// TIA Portal project "FactoryIO_Template_S7-1200_V16_V16" (V16)
// Vorlageprojekt für das Buch mit Zielsystem S7-1200

(* hardware
DEVICE "S7-1200-Station_1"  S7-1200 Station
   slot 0: "Baugruppenträger_0"  Rack  V1.0
   slot 1: "PLC_1"  CPU 1211C DC/DC/DC  6ES7 211-1AE40-0XB0  V4.1
*)

// ===== PLC "PLC_1"  CPU 1211C DC/DC/DC =====

VAR_GLOBAL   // PLC tag table "Standard-Variablentabelle"
   "START" AT %I0.0 : Bool;
   "STOP" AT %I0.1 : Bool;
   "V.S1" AT %I0.2 : Bool;
   "V.S4" AT %I0.3 : Bool;
   "V.S2" AT %I0.4 : Bool;
   "V.S3" AT %I0.5 : Bool;
   "BELT(6M)1" AT %Q0.0 : Bool;
   "BELT(2M)1" AT %Q0.1 : Bool;
   "BELLT(2M)2" AT %Q0.2 : Bool;
   "BELT(2M)3" AT %Q0.3 : Bool;
   "BELT(2M)4" AT %Q0.4 : Bool;
   "BELT CCW" AT %Q0.5 : Bool;
   "P1" AT %Q0.6 : Bool;
   "MOVE1" AT %Q0.7 : Bool;
   "P2" AT %Q1.0 : Bool;
   "MOVE2" AT %Q1.1 : Bool;
   "P3" AT %Q1.2 : Bool;
   "MOVE3" AT %Q1.3 : Bool;
   "MARKER" AT %M0.0 : Bool;
   "MARKER2" AT %M0.1 : Bool;
   "MARKER3" AT %M0.2 : Bool;
   "MARKER4" AT %M0.3 : Bool;
   "P1 MARKER" AT %M0.4 : Bool;
   "P3 MARKER" AT %M0.5 : Bool;
   "P2 MARKER" AT %M0.6 : Bool;
END_VAR

// folder: System blocks/Program resources

DATA_BLOCK "T1"   // DB1
{ S7_Optimized_Access := 'TRUE' }
AUTHOR : Simatic
FAMILY : IEC
NAME : IEC_TMR
VERSION : 1.0
// stored: InstanceOfName IEC_TIMER
"IEC_TIMER"
BEGIN
END_DATA_BLOCK

DATA_BLOCK "T2"   // DB2
{ S7_Optimized_Access := 'TRUE' }
AUTHOR : Simatic
FAMILY : IEC
NAME : IEC_TMR
VERSION : 1.0
// stored: InstanceOfName IEC_TIMER
"IEC_TIMER"
BEGIN
END_DATA_BLOCK

DATA_BLOCK "T3"   // DB3
{ S7_Optimized_Access := 'TRUE' }
AUTHOR : Simatic
FAMILY : IEC
NAME : IEC_TMR
VERSION : 1.0
// stored: InstanceOfName IEC_TIMER
"IEC_TIMER"
BEGIN
END_DATA_BLOCK

// folder: (top level)

FUNCTION "MHJ-PLC-Lab-Function-S71200" : Void   // FC9000, SCL
{ S7_Optimized_Access := 'TRUE' }
VERSION : 0.1
   VAR_TEMP
      rdTimeReturn : Int;
      outputTime : DTL;
      SyncVal : Byte;
      forVal : Int;
      forVal_2 : Int;
      Value : Byte;
   END_VAR
   VAR CONSTANT
      CompVal : Byte := 16#34;
      Value_01 : Byte := 16#11;
      Value_01_DW : DWord := 16#A165_D992;
      Value_02_DW : DWord := 16#58BE_4401;
   END_VAR
BEGIN

   #Value:=PEEK(area := 16#82,
        dbNumber := 0,
        byteOffset := 511);
   #Value := #Value + 1;

   POKE(area := 16#82,
        dbNumber := 0,
        byteOffset := 511,
        value := #Value);

   POKE(area:=16#81,
        dbNumber:=0,
        byteOffset:=1016,
        value:=#Value_01_DW);
   POKE(area := 16#81,
        dbNumber := 0,
        byteOffset := 1020,
        value := #Value_02_DW);

   POKE(area := 16#81,
        dbNumber := 0,
        byteOffset := 511,
        value := B#16#00);

   FOR #forVal := 0 TO 120 DO
       FOR #forVal_2:=0 TO 10 DO
           #rdTimeReturn:=RD_SYS_T(#outputTime);
           #rdTimeReturn := WR_SYS_T(#outputTime);
           #rdTimeReturn := RD_SYS_T(#outputTime);
           #rdTimeReturn := WR_SYS_T(#outputTime);
       END_FOR;
       #SyncVal:= PEEK(area := 16#81,
                      dbNumber := 0,
                      byteOffset := 511);
       IF #SyncVal = #CompVal THEN
          GOTO M_1;
       END_IF;
   END_FOR;
   RETURN;

   M_1:
   POKE(area := 16#81,
        dbNumber := 0,
        byteOffset := 511,
        value := B#16#0);
END_FUNCTION

ORGANIZATION_BLOCK "Main"   // OB1, LAD, ProgramCycle
TITLE = "Main Program Sweep (Cycle)"
{ S7_Optimized_Access := 'TRUE' }
VERSION : 0.1
   VAR_INPUT
      Initial_Call : Bool;   // Initial call of this OB
      Remanence : Bool;   // =True, if remanent data are available
   END_VAR
BEGIN

REGION Network 1: Konnektierungsbaustein für PLC-Lab
   // Im Netzwerk 1 wird der Konnektierungsbaustein für PLC-Lab aufgerufen.
   // Dieser Aufruf darf nicht entfernt werden!
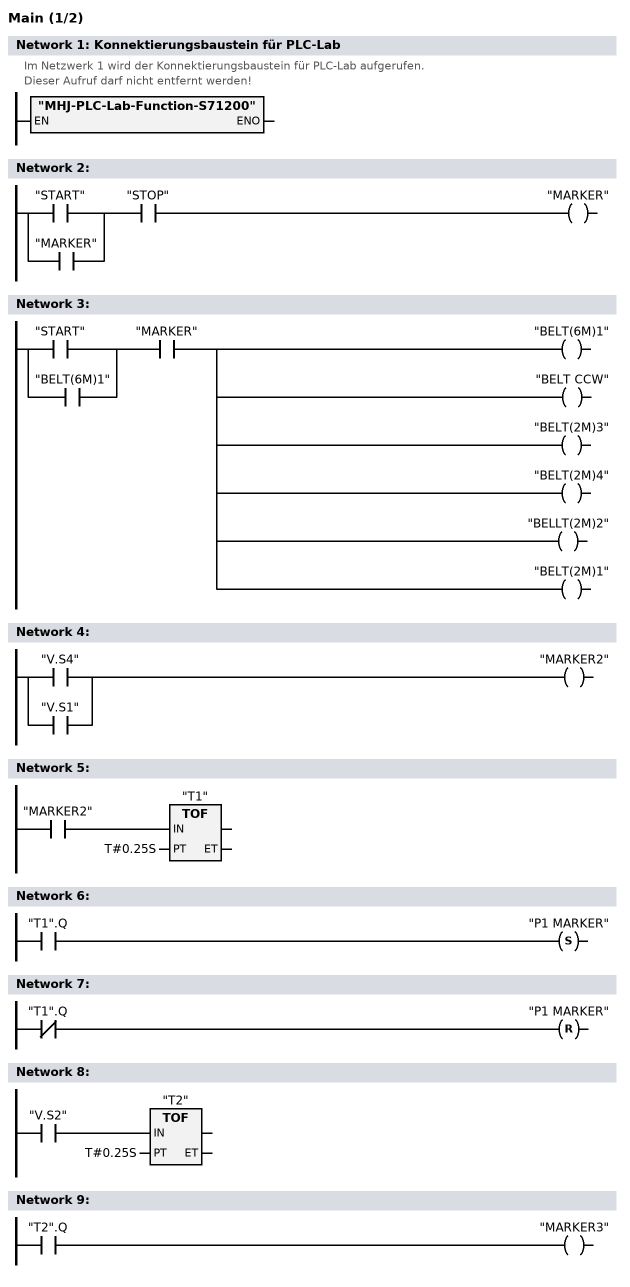
   RUNG wire#powerrail
      "MHJ-PLC-Lab-Function-S71200"()
   END_RUNG
   // the same network as SCL:
   "MHJ-PLC-Lab-Function-S71200"();
END_REGION

REGION Network 2
   RUNG wire#powerrail
      Contact( "START" )
      wire#w1
      Contact( "STOP" )
      Coil( "MARKER" )
   END_RUNG
   RUNG wire#powerrail
      Contact( "MARKER" )
   END_RUNG wire#w1
   // the same network as SCL:
   "MARKER" := ("START" OR "MARKER") AND "STOP";
END_REGION

REGION Network 3
   RUNG wire#powerrail
      Contact( "START" )
      wire#w1
      Contact( "MARKER" )
      wire#w2
      Coil( "BELT(6M)1" )
   END_RUNG
   RUNG wire#powerrail
      Contact( "BELT(6M)1" )
   END_RUNG wire#w1
   RUNG wire#w2
      Coil( "BELT CCW" )
   END_RUNG
   RUNG wire#w2
      Coil( "BELT(2M)3" )
   END_RUNG
   RUNG wire#w2
      Coil( "BELT(2M)4" )
   END_RUNG
   RUNG wire#w2
      Coil( "BELLT(2M)2" )
   END_RUNG
   RUNG wire#w2
      Coil( "BELT(2M)1" )
   END_RUNG
   // the same network as SCL:
   "BELT(6M)1" := ("START" OR "BELT(6M)1") AND "MARKER";
   "BELT CCW" := "BELT(6M)1";
   "BELT(2M)3" := "BELT(6M)1";
   "BELT(2M)4" := "BELT(6M)1";
   "BELLT(2M)2" := "BELT(6M)1";
   "BELT(2M)1" := "BELT(6M)1";
END_REGION

REGION Network 4
   RUNG wire#powerrail
      Contact( "V.S4" )
      wire#w1
      Coil( "MARKER2" )
   END_RUNG
   RUNG wire#powerrail
      Contact( "V.S1" )
   END_RUNG wire#w1
   // the same network as SCL:
   "MARKER2" := "V.S4" OR "V.S1";
END_REGION

REGION Network 5
   "T1".TOF(IN := "MARKER2", PT := T#0.25S);
END_REGION

REGION Network 6
   RUNG wire#powerrail
      Contact( "T1".Q )
      S_Coil( "P1 MARKER" )
   END_RUNG
   // the same network as SCL:
   IF "T1".Q THEN "P1 MARKER" := TRUE; END_IF;
END_REGION

REGION Network 7
   RUNG wire#powerrail
      I_Contact( "T1".Q )
      R_Coil( "P1 MARKER" )
   END_RUNG
   // the same network as SCL:
   IF NOT "T1".Q THEN "P1 MARKER" := FALSE; END_IF;
END_REGION

REGION Network 8
   "T2".TOF(IN := "V.S2", PT := T#0.25S);
END_REGION

REGION Network 9
   RUNG wire#powerrail
      Contact( "T2".Q )
      Coil( "MARKER3" )
   END_RUNG
   // the same network as SCL:
   "MARKER3" := "T2".Q;
END_REGION

REGION Network 10
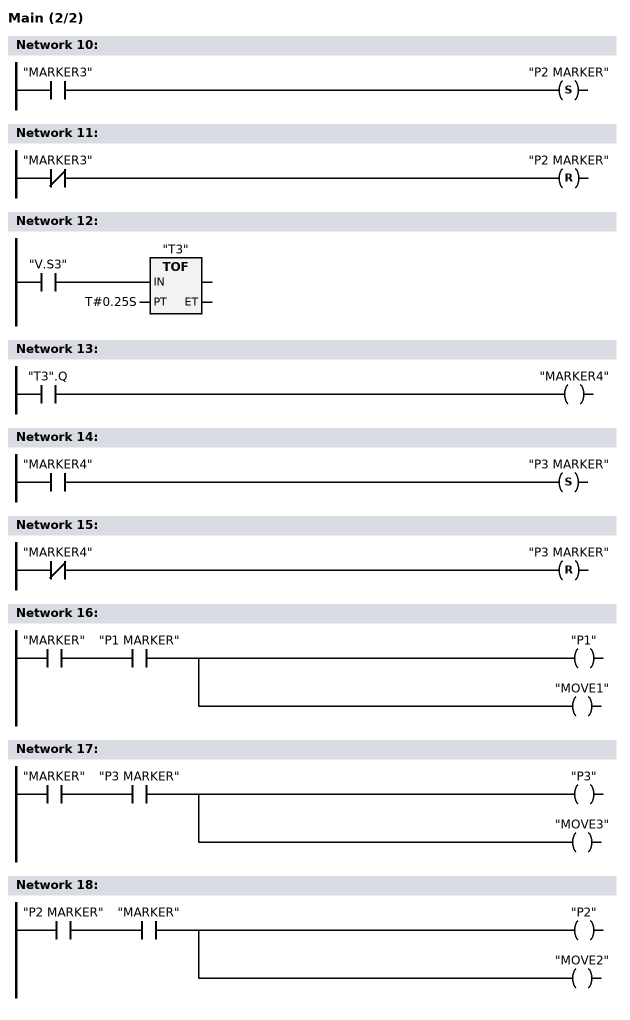
   RUNG wire#powerrail
      Contact( "MARKER3" )
      S_Coil( "P2 MARKER" )
   END_RUNG
   // the same network as SCL:
   IF "MARKER3" THEN "P2 MARKER" := TRUE; END_IF;
END_REGION

REGION Network 11
   RUNG wire#powerrail
      I_Contact( "MARKER3" )
      R_Coil( "P2 MARKER" )
   END_RUNG
   // the same network as SCL:
   IF NOT "MARKER3" THEN "P2 MARKER" := FALSE; END_IF;
END_REGION

REGION Network 12
   "T3".TOF(IN := "V.S3", PT := T#0.25S);
END_REGION

REGION Network 13
   RUNG wire#powerrail
      Contact( "T3".Q )
      Coil( "MARKER4" )
   END_RUNG
   // the same network as SCL:
   "MARKER4" := "T3".Q;
END_REGION

REGION Network 14
   RUNG wire#powerrail
      Contact( "MARKER4" )
      S_Coil( "P3 MARKER" )
   END_RUNG
   // the same network as SCL:
   IF "MARKER4" THEN "P3 MARKER" := TRUE; END_IF;
END_REGION

REGION Network 15
   RUNG wire#powerrail
      I_Contact( "MARKER4" )
      R_Coil( "P3 MARKER" )
   END_RUNG
   // the same network as SCL:
   IF NOT "MARKER4" THEN "P3 MARKER" := FALSE; END_IF;
END_REGION

REGION Network 16
   RUNG wire#powerrail
      Contact( "MARKER" )
      Contact( "P1 MARKER" )
      wire#w1
      Coil( "P1" )
   END_RUNG
   RUNG wire#w1
      Coil( "MOVE1" )
   END_RUNG
   // the same network as SCL:
   "P1" := "MARKER" AND "P1 MARKER";
   "MOVE1" := "P1";
END_REGION

REGION Network 17
   RUNG wire#powerrail
      Contact( "MARKER" )
      Contact( "P3 MARKER" )
      wire#w1
      Coil( "P3" )
   END_RUNG
   RUNG wire#w1
      Coil( "MOVE3" )
   END_RUNG
   // the same network as SCL:
   "P3" := "MARKER" AND "P3 MARKER";
   "MOVE3" := "P3";
END_REGION

REGION Network 18
   RUNG wire#powerrail
      Contact( "P2 MARKER" )
      Contact( "MARKER" )
      wire#w1
      Coil( "P2" )
   END_RUNG
   RUNG wire#w1
      Coil( "MOVE2" )
   END_RUNG
   // the same network as SCL:
   "P2" := "P2 MARKER" AND "MARKER";
   "MOVE2" := "P2";
END_REGION
END_ORGANIZATION_BLOCK